// TIA Portal V16 export
// export: Created 2026-04-03T07:27:29.8348699Z, ExportSetting WithDefaults, DisplayName Totally Integrated Automation Portal, DisplayVersion V16, DisplayName TIA Portal Version Control Interface, DisplayVersion V16, DisplayName TIA Portal Openness, DisplayVersion V16, DisplayName STEP 7 Professional, DisplayVersion V16, DisplayName STEP 7 Safety, DisplayVersion V16, DisplayName WinCC Advanced, DisplayVersion V16
FUNCTION "FC_Scale_Instance" : Void   // FC19, FBD
VERSION : 0.1
// stored: AutoNumber true, IsIECCheckEnabled false, UDAEnableTagReadback false
BEGIN

REGION Network 1
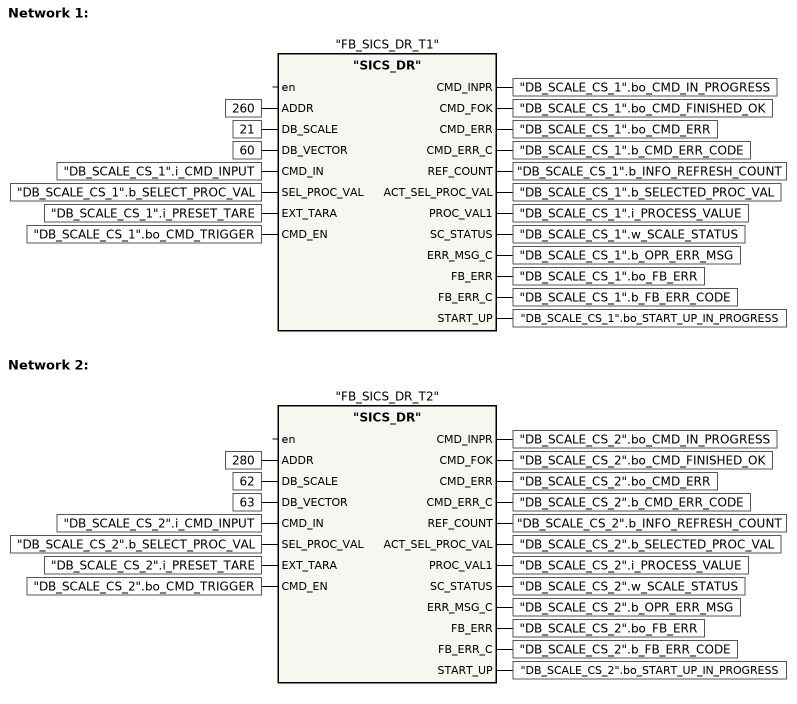
   "FB_SICS_DR_T1"(ADDR := 260,   // "SICS_DR"
                   DB_SCALE := 21,
                   DB_VECTOR := 60,
                   CMD_IN := "DB_SCALE_CS_1".i_CMD_INPUT,
                   SEL_PROC_VAL := "DB_SCALE_CS_1".b_SELECT_PROC_VAL,
                   EXT_TARA := "DB_SCALE_CS_1".i_PRESET_TARE,
                   CMD_EN := "DB_SCALE_CS_1".bo_CMD_TRIGGER,
                   CMD_INPR => "DB_SCALE_CS_1".bo_CMD_IN_PROGRESS,
                   CMD_FOK => "DB_SCALE_CS_1".bo_CMD_FINISHED_OK,
                   CMD_ERR => "DB_SCALE_CS_1".bo_CMD_ERR,
                   CMD_ERR_C => "DB_SCALE_CS_1".b_CMD_ERR_CODE,
                   REF_COUNT => "DB_SCALE_CS_1".b_INFO_REFRESH_COUNT,
                   ACT_SEL_PROC_VAL => "DB_SCALE_CS_1".b_SELECTED_PROC_VAL,
                   PROC_VAL1 => "DB_SCALE_CS_1".i_PROCESS_VALUE,
                   SC_STATUS => "DB_SCALE_CS_1".w_SCALE_STATUS,
                   ERR_MSG_C => "DB_SCALE_CS_1".b_OPR_ERR_MSG,
                   FB_ERR => "DB_SCALE_CS_1".bo_FB_ERR,
                   FB_ERR_C => "DB_SCALE_CS_1".b_FB_ERR_CODE,
                   START_UP => "DB_SCALE_CS_1".bo_START_UP_IN_PROGRESS);
END_REGION

REGION Network 2
   "FB_SICS_DR_T2"(ADDR := 280,   // "SICS_DR"
                   DB_SCALE := 62,
                   DB_VECTOR := 63,
                   CMD_IN := "DB_SCALE_CS_2".i_CMD_INPUT,
                   SEL_PROC_VAL := "DB_SCALE_CS_2".b_SELECT_PROC_VAL,
                   EXT_TARA := "DB_SCALE_CS_2".i_PRESET_TARE,
                   CMD_EN := "DB_SCALE_CS_2".bo_CMD_TRIGGER,
                   CMD_INPR => "DB_SCALE_CS_2".bo_CMD_IN_PROGRESS,
                   CMD_FOK => "DB_SCALE_CS_2".bo_CMD_FINISHED_OK,
                   CMD_ERR => "DB_SCALE_CS_2".bo_CMD_ERR,
                   CMD_ERR_C => "DB_SCALE_CS_2".b_CMD_ERR_CODE,
                   REF_COUNT => "DB_SCALE_CS_2".b_INFO_REFRESH_COUNT,
                   ACT_SEL_PROC_VAL => "DB_SCALE_CS_2".b_SELECTED_PROC_VAL,
                   PROC_VAL1 => "DB_SCALE_CS_2".i_PROCESS_VALUE,
                   SC_STATUS => "DB_SCALE_CS_2".w_SCALE_STATUS,
                   ERR_MSG_C => "DB_SCALE_CS_2".b_OPR_ERR_MSG,
                   FB_ERR => "DB_SCALE_CS_2".bo_FB_ERR,
                   FB_ERR_C => "DB_SCALE_CS_2".b_FB_ERR_CODE,
                   START_UP => "DB_SCALE_CS_2".bo_START_UP_IN_PROGRESS);
END_REGION
END_FUNCTION
